FUNCTION_BLOCK FB_Heater
VAR_INPUT
	bEnable 		: BOOL;	
	fHeatingSpeed 	: REAL := 1; //[*/s]
	fCoolingSpeed 	: REAL := 1; //[*/s]
	fLimitMin 		: REAL := 0; //[*]
	fLimitMax 		: REAL := 100; //[*]
END_VAR

VAR_OUTPUT
	bEnabled 		: BOOL;
	bIsLimitMin		: BOOL;
	bIsLimitMax		: BOOL;	
END_VAR

VAR
	_fValue 		: REAL; //[*]
END_VAR

InitRun();

bEnabled := bEnable;

_fValue := _fValue - fCoolingSpeed * GVL_Core.fbSystem.fDeltaTime;

IF bEnable THEN
	_fValue := _fValue + fHeatingSpeed * GVL_Core.fbSystem.fDeltaTime;
END_IF

bIsLimitMin := _fValue <= fLimitMin;
bIsLimitMax := _fValue >= fLimitMax;
_fValue := LIMIT(fLimitMin, _fValue, fLimitMax);

PROPERTY fValue : REAL
GET
fValue := _fValue;
END_GET
SET
_fValue := fValue;
END_SET
END_PROPERTY

METHOD INTERNAL InitRun
VAR_INST
	bInitRun : BOOL := TRUE;
END_VAR
IF NOT bInitRun THEN RETURN; END_IF
bInitRun := FALSE;
END_METHOD

END_FUNCTION_BLOCK

(* stored: Version 1.1.0.1, ProductVersion 3.1.4024.12
   POU FB_Heater: Id {e09e2890-7221-0f07-0e61-61432d4b0f35}, SpecialFunc None
   Property fValue: Id {0964f444-8c81-0f60-0117-e0741ceae9eb}
   Get Get: Id {b7eba905-2b22-01db-2ca3-08b0ab0d9f8e}
   Set Set: Id {5387611c-2a16-0f90-31f6-08be77052067}
   Method InitRun: Id {c92c38b6-adc3-0282-245f-9e2f7faaa523} *)
